FUNCTION_BLOCK W3W4 (* Basic Function Block Type *)
  (* Standard: 61499-2 *)
  (* Version 0.0, 9/24/2018, dmidro, nxtControl GmbH, Template *)
  PACKAGE Main;
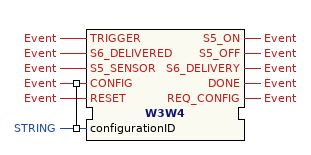
  EVENT_INPUT
    TRIGGER;
    S6_DELIVERED;
    S5_SENSOR;
    CONFIG WITH configurationID;
    RESET;
  END_EVENT
  EVENT_OUTPUT
    S5_ON;
    S5_OFF;
    S6_DELIVERY;
    DONE;
    REQ_CONFIG;
  END_EVENT
  VAR_INPUT
    configurationID : STRING;
  END_VAR
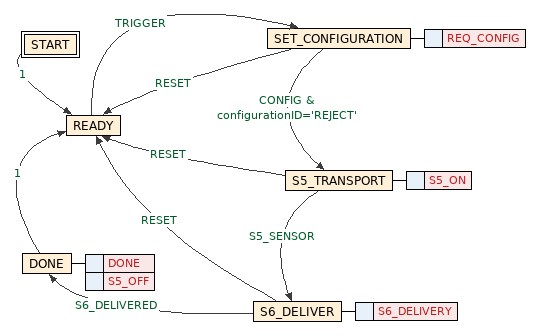
  EC_STATES
    START; (* Initial State *)
    S5_TRANSPORT : -> S5_ON;
    S6_DELIVER : -> S6_DELIVERY;
    DONE : -> DONE, -> S5_OFF;
    READY;
    SET_CONFIGURATION : -> REQ_CONFIG;
  END_STATES
  EC_TRANSITIONS
    START TO READY := 1;
    S5_TRANSPORT TO S6_DELIVER := S5_SENSOR;
    S6_DELIVER TO DONE := S6_DELIVERED;
    READY TO SET_CONFIGURATION := TRIGGER;
    SET_CONFIGURATION TO S5_TRANSPORT := CONFIG & configurationID='REJECT';
    DONE TO READY := 1;
    SET_CONFIGURATION TO READY := RESET;
    S5_TRANSPORT TO READY := RESET;
    S6_DELIVER TO READY := RESET;
  END_TRANSITIONS
  ALGORITHM INIT IN ST: (* Initialization algorithm *)
;
  END_ALGORITHM
  ALGORITHM REQ IN ST: (* Normally executed algorithm *)
;
  END_ALGORITHM
END_FUNCTION_BLOCK
